Universal Robots PolyScope program: mpc.urp

Program mpc (installation=default directory=/programs createdIn=5.11.9.1010452 lastSavedIn=5.11.9.1010452 robotSerialNumber=20225200364)
Calibrated DH parameters: a=[0.00002, -0.569483, -0.54992, -0.00001, -0.000036, 0]; d=[0.180894, -146.691669, 192.918669, -46.053088, 0.119778, 0.115602]; alpha=[1.571425, -0.001534, 0.003359, 1.568739, -1.571477, 0]; deltaTheta=[0, 0.376258, -0.101074, -0.275185, -0.000002, 0]
Robot Program (runOnlyOnce=false)
  URCap RG Grip (OnRobot, OnRobot A/S) dataModel(workpiece-lost=false, rg-target-width=0.04, rg-target-force=26.0, Variable(key=on_return, variable(name=on_return)))
  MoveJ speed 0.5 deg/s, acceleration 0.5 deg/s^2 (useActiveTCP=true) feature=Base
    Waypoint Waypoint_1: TCP in base x=369.435 y=295.335 z=147.109 mm, rx=1.7125 ry=-0.0436 rz=0.0435 rad; joints [66.364, -135.849, -123.922, -271.445, -66.65, -180.27] deg
    MoveJ speed 0.5 deg/s, acceleration 0.5 deg/s^2 (useActiveTCP=true) feature=Base
      Waypoint Waypoint_2: TCP in base x=369.428 y=209.517 z=147.157 mm, rx=1.7127 ry=-0.0437 rz=0.0436 rad; joints [62.021, -134.863, -130.584, -265.453, -62.366, -180.998] deg
